FUNCTION_BLOCK XtsPart EXTENDS CyclicBase
VAR
	_MyInterface : Tc3_XTS_Utility.I_TcIoXtsXpuPart;
	XtsIoEnvInitialiseState : INT;
	MyModuleCount : UDINT;
	PartDriveState: Tc3_XTS_Utility.DriveState;
	_ReadyToEnable: BOOL;
	MyModules : ARRAY[0..SystemParameters.MaxModulesInPart] OF XtsMotorModule;
	ModuleIndex: UDINT := 1;
	InSim : BOOL;
	i : UINT;
END_VAR

METHOD PUBLIC  Cycle : HRESULT
VAR_INPUT
END_VAR
PartDriveState := _MyInterface.GetDriveState();

CASE PartDriveState OF
	DriveState.Unknown:
		_ReadyToEnable := FALSE;

	DriveState.FaultReactionActive:
		_ReadyToEnable := FALSE;

	DriveState.Fault:
		_ReadyToEnable := FALSE;

	DriveState.NotReadyToSwitchOn:
		_ReadyToEnable := FALSE;

	DriveState.SwitchOnDisabled:
		_ReadyToEnable := FALSE;

	DriveState.ReadyToSwitchOn:
		_ReadyToEnable := TRUE;

	DriveState.SwitchedOn:
		_ReadyToEnable := TRUE;

	DriveState.OperationEnabled:
		_ReadyToEnable := TRUE;

ELSE
	_ReadyToEnable := FALSE;
END_CASE

FOR i := 0 TO (UDINT_TO_UINT(MyModuleCount) - 1) DO
	MyModules[i].Cycle();
END_FOR
END_METHOD

METHOD Initialise : HRESULT
VAR_INPUT
END_VAR
CASE XtsIoEnvInitialiseState OF
	0:
		IF _MyInterface <> 0 THEN
			XtsIoEnvInitialiseState := 1;
		ELSE
			XtsIoEnvInitialiseState := 999;
		END_IF
	1:
		MyModuleCount := _MyInterface.GetModuleCount();
		IF InSim THEN
			XtsIoEnvInitialiseState := 3;
			FOR i := 0 TO UDINT_TO_UINT(MyModuleCount - 1) DO
				MyModules[i].SetInSim();
			END_FOR
			InSim := true;
		ELSE
			FOR i := 0 TO UDINT_TO_UINT(MyModuleCount - 1) DO
				MyModules[i].MyCoEInterface := _MyInterface.ModuleCoE(i + 1);
				MyModules[i].MyModuleInterface := _MyInterface.ModuleTcIo(i + 1);
			END_FOR
			XtsIoEnvInitialiseState := 2;
		END_IF
		
	2:
		XtsIoEnvInitialiseState := 3;
		FOR i := 0 TO UDINT_TO_UINT(MyModuleCount-1) DO
			IF MyModules[i].Initialise() <> 2 THEN
				XtsIoEnvInitialiseState := 2;
			END_IF
		END_FOR
	3:
		Initialise := 2;

END_CASE
END_METHOD

METHOD Is24VBusOK : BOOL
VAR_INPUT
END_VAR
Is24VBusOK := TRUE;
FOR i := 0 TO (UDINT_TO_UINT(MyModuleCount) - 1) DO
	IF MyModules[i].Is24VOK() = 1 THEN
		Is24VBusOK := FALSE;
	END_IF
END_FOR
END_METHOD

METHOD Is48VBusOK : BOOL
VAR_INPUT
END_VAR
Is48VBusOK := TRUE;
FOR i := 0 TO (UDINT_TO_UINT(MyModuleCount) - 1) DO
	IF MyModules[i].Is48VOK() = 1 THEN
		Is48VBusOK := FALSE;
	END_IF
END_FOR
END_METHOD

PROPERTY MyXtsIoEnvInterface : I_TcIoXtsXpuPart
GET
MyXtsIoEnvInterface := _MyInterface;
END_GET
SET
_MyInterface := MyXtsIoEnvInterface;
END_SET
END_PROPERTY

METHOD ResetPart : BOOL
VAR_INPUT
END_VAR
ResetPart := _MyInterface.TriggerReset();
END_METHOD

METHOD SetInSim : HRESULT
VAR_INPUT
END_VAR
InSim := true;
END_METHOD

END_FUNCTION_BLOCK

(* stored: Version 1.1.0.1
   POU XtsPart: Id {39541d00-22ec-4750-829d-4864a624597e}, SpecialFunc None
   Method Cycle: Id {6aa26807-846b-4168-ab87-fb4c66b138eb}
   Method Initialise: Id {f7bcb601-a320-4f3f-bcf3-5ec4e45a7245}
   Method Is24VBusOK: Id {d79d6eda-1f90-4384-9dda-ac7f4aaa7f07}
   Method Is48VBusOK: Id {44113d88-367f-494b-87cf-4655fd94d258}
   Property MyXtsIoEnvInterface: Id {b5f6c838-c909-4a11-9656-9e449699aee4}
   Get Get: Id {249dae7e-fa2b-4c2d-a421-a33d92e9b50d}
   Set Set: Id {436f8d77-48c4-4edc-81e4-5821f3038a93}
   Method ResetPart: Id {a2c1bf74-a00f-4e37-abd0-e53201644a52}
   Method SetInSim: Id {273102d0-bbf8-41a5-af45-2632119808d5} *)
